ABB RAPID module: Module1.mod

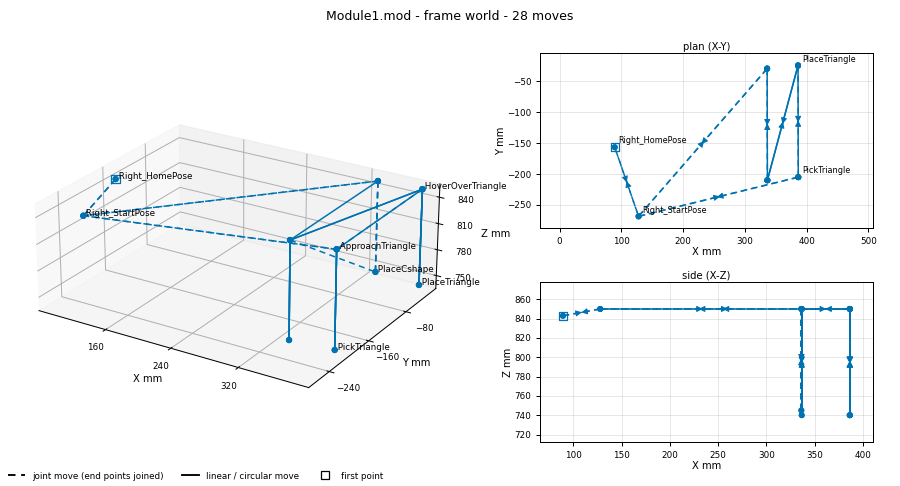
[picture p0: tool path of Module1.mod in frame world, 28 of 28 moves have a stored position in this frame; points joined in program order, loops and branches not executed]
MODULE Module1
    CONST robtarget Right_HomePose:=[[89.387946422,-156.622117956,842.913470217],[0.066010726,-0.842420918,-0.111214912,-0.523068661],[0,0,0,4],[-101.964427132,9E+09,9E+09,9E+09,9E+09,9E+09]];
    CONST robtarget Right_StartPose:=[[127.970106572,-268.540442898,849.999919372],[0.110773358,0.282535603,0.887093552,0.347804438],[0,0,0,4],[-91.873037584,9E+09,9E+09,9E+09,9E+09,9E+09]];
    CONST robtarget ApproachTriangle:=[[0,0,100],[0,0,0.923879533,0.382683432],[0,-1,0,4],[-90.504149971,9E+09,9E+09,9E+09,9E+09,9E+09]];
    CONST robtarget PickTriangle:=[[0,0,-10],[0,0,0.923879533,0.382683432],[1,-1,0,4],[-90.504149971,9E+09,9E+09,9E+09,9E+09,9E+09]];
    CONST robtarget HoverOverTriangle:=[[24.71,-24.35,130],[0,0,0.923879533,0.382683432],[1,-1,0,4],[-90.504149971,9E+09,9E+09,9E+09,9E+09,9E+09]];
    CONST robtarget PlaceTriangle:=[[24.71,-24.35,20],[0,0,0.923879533,0.382683432],[1,-1,0,4],[-90.504149971,9E+09,9E+09,9E+09,9E+09,9E+09]];
    CONST robtarget ApproachCshape:=[[0,0,100],[0,0,0.923879533,0.382683432],[1,-1,0,4],[-90.504149971,9E+09,9E+09,9E+09,9E+09,9E+09]];
    CONST robtarget PickCshape:=[[0,0,-10],[0,0,0.923879533,0.382683432],[1,-1,0,4],[-90.504149971,9E+09,9E+09,9E+09,9E+09,9E+09]];
    CONST robtarget HoverOverCshape:=[[-25.29,-29.351,130],[0,0,0.923879533,0.382683432],[1,-1,2,4],[-90.504149971,9E+09,9E+09,9E+09,9E+09,9E+09]];
    CONST robtarget PlaceCshape:=[[-25.29,-29.351,25],[0,0,0.923879533,0.382683432],[1,-1,-2,4],[-90.504149971,9E+09,9E+09,9E+09,9E+09,9E+09]];
    PROC Path_10()
        ConfJ\Off;
        ConfL\Off;
        MoveJ Right_HomePose,v100,fine,Servo\WObj:=RightArm;
        MoveJ Right_StartPose,v100,fine,Servo\WObj:=RightArm;
        MoveJ ApproachTriangle,v100,fine,Servo\WObj:=TriangleObj;
        MoveL PickTriangle,v100,fine,Servo\WObj:=TriangleObj;
        g_GripIn;
        WaitTime 1;
        MoveL ApproachTriangle,v100,fine,Servo\WObj:=TriangleObj;
        MoveL HoverOverTriangle,v100,fine,Servo\WObj:=RightMainHolder;
        MoveL PlaceTriangle,v100,fine,Servo\WObj:=RightMainHolder;
        g_GripOut;
        WaitTime 1;
        MoveL HoverOverTriangle,v100,fine,Servo\WObj:=RightMainHolder;
        MoveL ApproachCshape,v100,fine,Servo\WObj:=CshapeObj;
        MoveL PickCshape,v100,fine,Servo\WObj:=CshapeObj;
        g_GripIn;
        WaitTime 1;
        MoveL ApproachCshape,v100,fine,Servo\WObj:=CshapeObj;
        MoveJ PlaceCshape,v100,fine,Servo\WObj:=RightMainHolder;
        g_GripOut;
        WaitTime 1;
        MoveJ HoverOverCshape,v100,fine,Servo\WObj:=RightMainHolder;
        MoveJ Right_StartPose,v100,fine,Servo\WObj:=RightArm;
        MoveJ HoverOverCshape,v100,fine,Servo\WObj:=RightMainHolder;
        MoveJ PlaceCshape,v100,fine,Servo\WObj:=RightMainHolder;
        g_GripIn;
        WaitTime 1;
        MoveJ HoverOverCshape,v100,fine,Servo\WObj:=RightMainHolder;
        MoveL ApproachCshape,v100,fine,Servo\WObj:=CshapeObj;
        MoveL PickCshape,v100,fine,Servo\WObj:=CshapeObj;
        g_GripOut;
        WaitTime 1;
        MoveL ApproachCshape,v100,fine,Servo\WObj:=CshapeObj;
        MoveL HoverOverTriangle,v100,fine,Servo\WObj:=RightMainHolder;
        MoveL PlaceTriangle,v100,fine,Servo\WObj:=RightMainHolder;
        g_GripIn;
        WaitTime 1;
        MoveL HoverOverTriangle,v100,fine,Servo\WObj:=RightMainHolder;
        MoveJ ApproachTriangle,v100,fine,Servo\WObj:=TriangleObj;
        MoveL PickTriangle,v100,fine,Servo\WObj:=TriangleObj;
        g_GripOut;
        WaitTime 1;
        MoveL ApproachTriangle,v100,fine,Servo\WObj:=TriangleObj;
        MoveJ Right_StartPose,v100,fine,Servo\WObj:=RightArm;
        MoveJ Right_HomePose,v100,fine,Servo\WObj:=RightArm;
    ENDPROC
ENDMODULE
